TYPE sGeneralState :
STRUCT
	boReady: BOOL;
	boCharging: BOOL;
	strPosition: STRING;
END_STRUCT
END_TYPE

(* stored: Version 1.1.0.1, ProductVersion 3.1.4026.13
   DUT sGeneralState: Id {ae4af2a2-ceab-46ee-a1c3-98a6ecb21365} *)
